(*
Casts I_Arg to I_Components
*)
FUNCTION IArgAsIComp : Result
VAR_INPUT
	iSource	: I_Arg;
END_VAR
VAR_OUTPUT
	iDest	: I_Component;
END_VAR

IF iSource = 0 THEN
	IArgAsIComp := Err.Itf0;
	RETURN;
END_IF

IF __QUERYINTERFACE(iSource, iDest) THEN
	IArgAsIComp := Ok;
ELSE
	iDest := 0;
	IArgAsIComp := Err.NoMatch;
END_IF

END_FUNCTION

(* stored: Version 1.1.0.1
   POU IArgAsIComp: Id {5c29e6e1-73d7-4b4a-82c7-dcd0d4c36bbf}, SpecialFunc None *)
